FUNCTION_BLOCK helperOutputSelection
VAR_INPUT
END_VAR
VAR_OUTPUT
END_VAR
VAR
	outputs AT%Q*: ARRAY[0..3] OF BOOL;
	
	nCounter : INT;
END_VAR

ACTION ReleaseAll:
FOR nCounter:=0 TO 3 BY 1 DO
	outputs[nCounter] := false;
END_FOR
END_ACTION

METHOD Trigger : BOOL
VAR_INPUT
	sensorPair : defSensorPair;
	state : BOOL; //ON/OFF
END_VAR
VAR
	index : BYTE;
END_VAR
index.0 := sensorPair.bit0;
index.1 := sensorPair.bit0;

outputs[index] := state;
END_METHOD

END_FUNCTION_BLOCK

(* stored: Version 1.1.0.1, ProductVersion 3.1.4024.0
   POU helperOutputSelection: Id {f971eeb7-afdd-4ea0-9e5c-3402194a0dc0}, SpecialFunc None
   Action ReleaseAll: Id {72b535c6-d0d2-4d16-8572-ca70d0a5ff1a}
   Method Trigger: Id {2643e95e-1bb4-40d4-aac8-7134c47d1fe2} *)
